{attribute 'qualified_only'}
{attribute 'strict'}
{attribute 'to_string'}
TYPE E_State :
(
	INIT:=0,
	EnableMover,
	EnableCheck,
	Zmove,
	ZmoveCheck,
	AddToGroup,
	AddToGroupCheck,
	EnableComp,
	DisableMover,
	DisableCheck,
	DisableComp,
	ERROR
);
END_TYPE

(* stored: Version 1.1.0.1
   DUT E_State: Id {0f0b0606-c0aa-4d5c-a291-238893cbf30b} *)
